// TIA Portal V16 export
// export: Created 2021-11-12T13:31:02.9636744Z, ExportSetting WithDefaults, DisplayName Totally Integrated Automation Portal, DisplayVersion V16 Update 3, DisplayName TIA Portal Version Control Interface, DisplayVersion V16 Update 2, DisplayName TIA Portal Openness, DisplayVersion V16 Update 3, DisplayName SINAMICS Startdrive Advanced, DisplayVersion V16 Update 5, DisplayName SINAMICS Startdrive G130, G150, S120, S150, SINAMICS MV, S210, DisplayVersion V16 Update 5, DisplayName SINAMICS Startdrive G110M, G120, G120C, G120D, G120P, G115D, DisplayVersion V16 Update 5, DisplayName STEP 7 Professional, DisplayVersion V16 Update 3, DisplayName STEP 7 Safety, DisplayVersion V16, DisplayName WinCC UA Professional, DisplayVersion V16 Update 3
FUNCTION_BLOCK "DataColl"   // FB65, LAD
TITLE = Data Collector for SCADA
{ S7_Optimized_Access := 'TRUE' }
VERSION : 0.1
// stored: AutoNumber true, IsIECCheckEnabled false, IsRetainMemResEnabled false, MemoryReserve 100, SetENOAutomatically false, UDAEnableTagReadback false
   VAR
      SS_Edge : Array[0..9] of Bool;
      SF_ArchivePeriodicallyFullAlarm : "STD_DI_Mon";
      SF_ArchivePeriodicallyFullWarn : "STD_DI_Mon";
      SF_ArchiveItemFullAlarm : "STD_DI_Mon";
      SF_ArchiveItemFullWarn : "STD_DI_Mon";
      SF_FIFOQueueArchivePeriodically : "FIFOQueueArchivPeriodically";   // FIFO for data collected periodically
      SF_FIFOQueueArchiveItem : "FIFOQueueArchivItem";   // FIFO for data collected on trigger
      SI_PointerArchivePeriodically : Int;   // Pointer in FIFO
      SI_PointerArchiveItem : Int;   // Pointer in FIFo
      SB1_BufferArchivePeriodicallyFullAlarm : Bool;   // Buffer full alarm
      SB1_BufferArchivePeriodicallyFullWarn : Bool;   // Buffer full warning
      SB1_BufferArchiveItemFullAlarm : Bool;   // Buffer full alarm
      SB1_BufferArchiveItemFullWarn : Bool;   // Buffer full warning
   END_VAR
   VAR_TEMP
      TB1CmdReader_ArchivePeriodically : Bool;   // Command to write data into FIFO
      TB1CmdReader_ArchiveItem1 : Bool;   // Command to write data into FIFO
      TB1CmdReader_ArchiveItem2 : Bool;   // Command to write data into FIFO
      TB1ArchiveItemDone : Bool;   // Writing data to FIFO done
      TB1EnableArchivePeriodically : Bool;   // Enable to archive data periodically
      TI_ArchiveLenght : Int;
   END_VAR
   VAR_TEMP   // added for the SCL form of the ladder/FBD networks
      _w1 : Bool;
      _w2 : Bool;
   END_VAR
BEGIN

REGION Network 1: Clear temporary variables
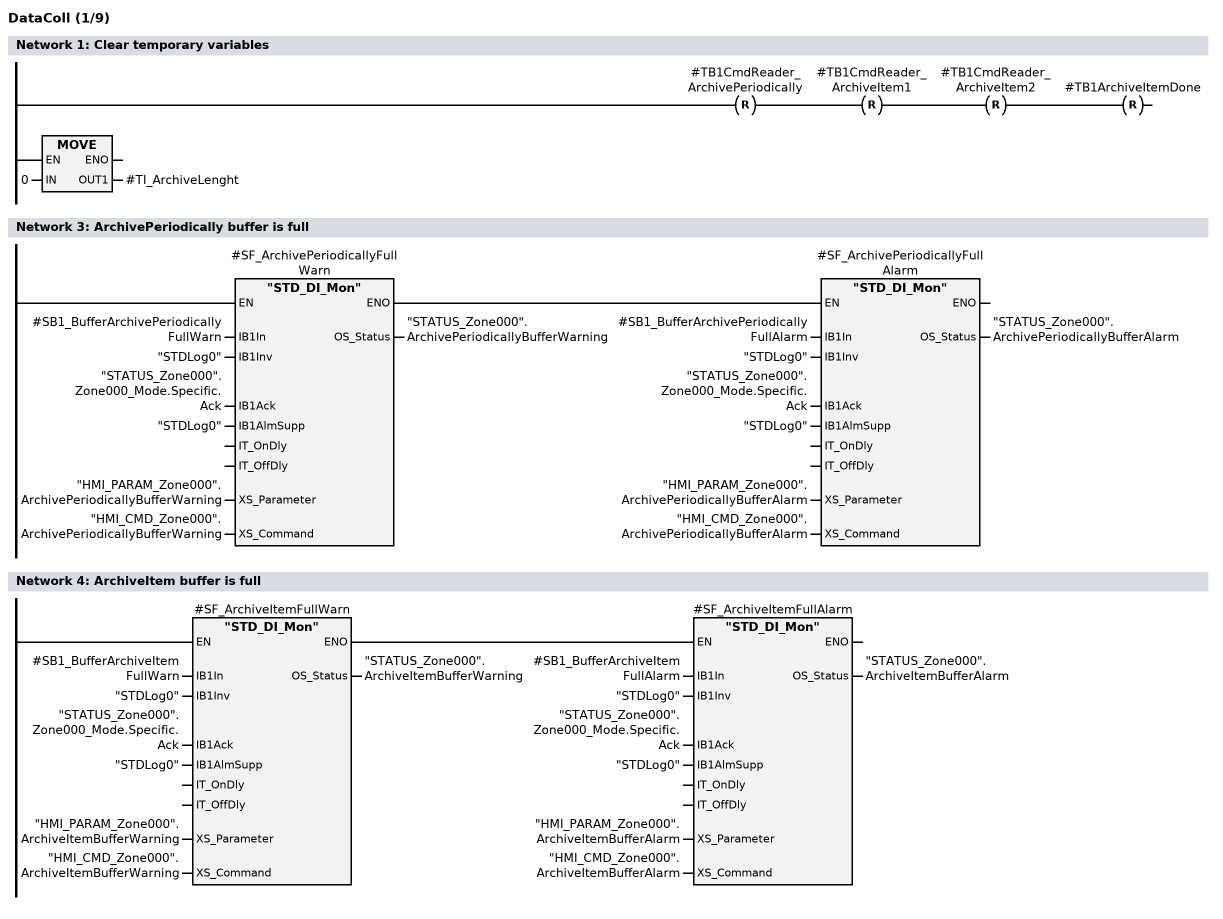
   RUNG wire#powerrail
      R_Coil( #TB1CmdReader_ArchivePeriodically )
      R_Coil( #TB1CmdReader_ArchiveItem1 )
      R_Coil( #TB1CmdReader_ArchiveItem2 )
      R_Coil( #TB1ArchiveItemDone )
   END_RUNG
   RUNG wire#powerrail
      Move(in := 0, out1 => #TI_ArchiveLenght)
   END_RUNG
   // the same network as SCL:
   #TB1CmdReader_ArchivePeriodically := FALSE;
   #TB1CmdReader_ArchiveItem1 := FALSE;
   #TB1CmdReader_ArchiveItem2 := FALSE;
   #TB1ArchiveItemDone := FALSE;
   #TI_ArchiveLenght := 0;
END_REGION

REGION Network 2: *************** Alarms ***************
END_REGION

REGION Network 3: ArchivePeriodically buffer is full
   RUNG wire#powerrail
      #SF_ArchivePeriodicallyFullWarn(IB1In := #SB1_BufferArchivePeriodicallyFullWarn, IB1Inv := "STDLog0", IB1Ack := "STATUS_Zone000".Zone000_Mode.Specific.Ack, IB1AlmSupp := "STDLog0", IT_OnDly :=, IT_OffDly :=, XS_Parameter := "HMI_PARAM_Zone000".ArchivePeriodicallyBufferWarning, XS_Command := "HMI_CMD_Zone000".ArchivePeriodicallyBufferWarning, OS_Status => "STATUS_Zone000".ArchivePeriodicallyBufferWarning)
      #SF_ArchivePeriodicallyFullAlarm(IB1In := #SB1_BufferArchivePeriodicallyFullAlarm, IB1Inv := "STDLog0", IB1Ack := "STATUS_Zone000".Zone000_Mode.Specific.Ack, IB1AlmSupp := "STDLog0", IT_OnDly :=, IT_OffDly :=, XS_Parameter := "HMI_PARAM_Zone000".ArchivePeriodicallyBufferAlarm, XS_Command := "HMI_CMD_Zone000".ArchivePeriodicallyBufferAlarm, OS_Status => "STATUS_Zone000".ArchivePeriodicallyBufferAlarm)
   END_RUNG
   // the same network as SCL:
   #SF_ArchivePeriodicallyFullWarn(IB1In := #SB1_BufferArchivePeriodicallyFullWarn,   // "STD_DI_Mon"
                           IB1Inv := "STDLog0",
                           IB1Ack := "STATUS_Zone000".Zone000_Mode.Specific.Ack,
                           IB1AlmSupp := "STDLog0",
                           XS_Parameter := "HMI_PARAM_Zone000".ArchivePeriodicallyBufferWarning,
                           XS_Command := "HMI_CMD_Zone000".ArchivePeriodicallyBufferWarning,
                           OS_Status => "STATUS_Zone000".ArchivePeriodicallyBufferWarning,
                           ENO => #_w1);
   IF #_w1 THEN
       #SF_ArchivePeriodicallyFullAlarm(IB1In := #SB1_BufferArchivePeriodicallyFullAlarm,   // "STD_DI_Mon"
                               IB1Inv := "STDLog0",
                               IB1Ack := "STATUS_Zone000".Zone000_Mode.Specific.Ack,
                               IB1AlmSupp := "STDLog0",
                               XS_Parameter := "HMI_PARAM_Zone000".ArchivePeriodicallyBufferAlarm,
                               XS_Command := "HMI_CMD_Zone000".ArchivePeriodicallyBufferAlarm,
                               OS_Status => "STATUS_Zone000".ArchivePeriodicallyBufferAlarm);
   END_IF;
END_REGION

REGION Network 4: ArchiveItem buffer is full
   RUNG wire#powerrail
      #SF_ArchiveItemFullWarn(IB1In := #SB1_BufferArchiveItemFullWarn, IB1Inv := "STDLog0", IB1Ack := "STATUS_Zone000".Zone000_Mode.Specific.Ack, IB1AlmSupp := "STDLog0", IT_OnDly :=, IT_OffDly :=, XS_Parameter := "HMI_PARAM_Zone000".ArchiveItemBufferWarning, XS_Command := "HMI_CMD_Zone000".ArchiveItemBufferWarning, OS_Status => "STATUS_Zone000".ArchiveItemBufferWarning)
      #SF_ArchiveItemFullAlarm(IB1In := #SB1_BufferArchiveItemFullAlarm, IB1Inv := "STDLog0", IB1Ack := "STATUS_Zone000".Zone000_Mode.Specific.Ack, IB1AlmSupp := "STDLog0", IT_OnDly :=, IT_OffDly :=, XS_Parameter := "HMI_PARAM_Zone000".ArchiveItemBufferAlarm, XS_Command := "HMI_CMD_Zone000".ArchiveItemBufferAlarm, OS_Status => "STATUS_Zone000".ArchiveItemBufferAlarm)
   END_RUNG
   // the same network as SCL:
   #SF_ArchiveItemFullWarn(IB1In := #SB1_BufferArchiveItemFullWarn,   // "STD_DI_Mon"
                           IB1Inv := "STDLog0",
                           IB1Ack := "STATUS_Zone000".Zone000_Mode.Specific.Ack,
                           IB1AlmSupp := "STDLog0",
                           XS_Parameter := "HMI_PARAM_Zone000".ArchiveItemBufferWarning,
                           XS_Command := "HMI_CMD_Zone000".ArchiveItemBufferWarning,
                           OS_Status => "STATUS_Zone000".ArchiveItemBufferWarning,
                           ENO => #_w1);
   IF #_w1 THEN
       #SF_ArchiveItemFullAlarm(IB1In := #SB1_BufferArchiveItemFullAlarm,   // "STD_DI_Mon"
                               IB1Inv := "STDLog0",
                               IB1Ack := "STATUS_Zone000".Zone000_Mode.Specific.Ack,
                               IB1AlmSupp := "STDLog0",
                               XS_Parameter := "HMI_PARAM_Zone000".ArchiveItemBufferAlarm,
                               XS_Command := "HMI_CMD_Zone000".ArchiveItemBufferAlarm,
                               OS_Status => "STATUS_Zone000".ArchiveItemBufferAlarm);
   END_IF;
END_REGION

REGION Network 5: ************** Data collecting on trigger ***************
END_REGION

REGION Network 6: Filling interface for item1
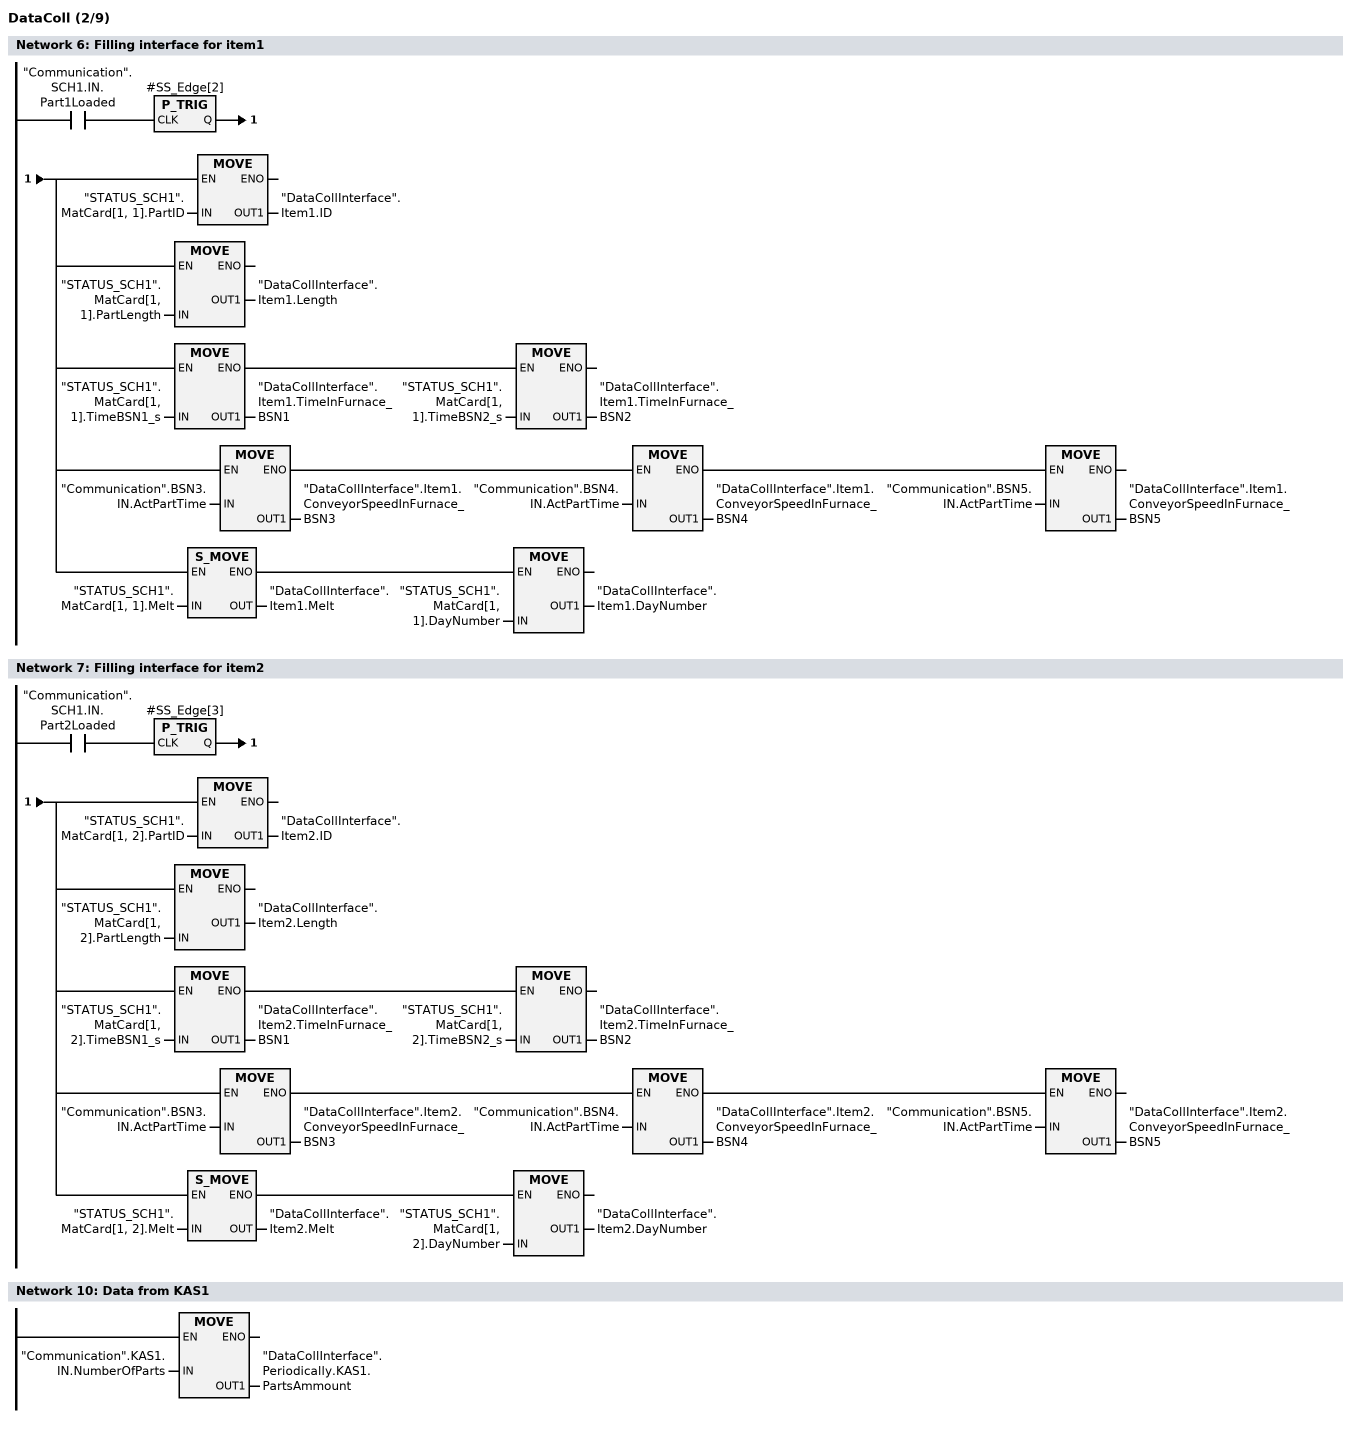
   RUNG wire#powerrail
      Contact( "Communication".SCH1.IN.Part1Loaded )
      P_Trig( #SS_Edge[2] )
      wire#w1
      Move(in := "STATUS_SCH1".MatCard[1, 1].PartID, out1 => "DataCollInterface".Item1.ID)
   END_RUNG
   RUNG wire#w1
      Move(in := "STATUS_SCH1".MatCard[1, 1].PartLength, out1 => "DataCollInterface".Item1.Length)
   END_RUNG
   RUNG wire#w1
      Move(in := "STATUS_SCH1".MatCard[1, 1].TimeBSN1_s, out1 => "DataCollInterface".Item1.TimeInFurnace_BSN1)
      Move(in := "STATUS_SCH1".MatCard[1, 1].TimeBSN2_s, out1 => "DataCollInterface".Item1.TimeInFurnace_BSN2)
   END_RUNG
   RUNG wire#w1
      Move(in := "Communication".BSN3.IN.ActPartTime, out1 => "DataCollInterface".Item1.ConveyorSpeedInFurnace_BSN3)
      Move(in := "Communication".BSN4.IN.ActPartTime, out1 => "DataCollInterface".Item1.ConveyorSpeedInFurnace_BSN4)
      Move(in := "Communication".BSN5.IN.ActPartTime, out1 => "DataCollInterface".Item1.ConveyorSpeedInFurnace_BSN5)
   END_RUNG
   RUNG wire#w1
      S_Move(in := "STATUS_SCH1".MatCard[1, 1].Melt, out => "DataCollInterface".Item1.Melt)
      Move(in := "STATUS_SCH1".MatCard[1, 1].DayNumber, out1 => "DataCollInterface".Item1.DayNumber)
   END_RUNG
   // the same network as SCL:
   #_w1 := "Communication".SCH1.IN.Part1Loaded AND NOT #SS_Edge[2];   // rising edge
   #SS_Edge[2] := "Communication".SCH1.IN.Part1Loaded;
   IF #_w1 THEN
       "DataCollInterface".Item1.ID := "STATUS_SCH1".MatCard[1, 1].PartID;
       "DataCollInterface".Item1.Length := "STATUS_SCH1".MatCard[1, 1].PartLength;
       "DataCollInterface".Item1.TimeInFurnace_BSN1 := "STATUS_SCH1".MatCard[1, 1].TimeBSN1_s;
       "DataCollInterface".Item1.TimeInFurnace_BSN2 := "STATUS_SCH1".MatCard[1, 1].TimeBSN2_s;
       "DataCollInterface".Item1.ConveyorSpeedInFurnace_BSN3 := "Communication".BSN3.IN.ActPartTime;
       "DataCollInterface".Item1.ConveyorSpeedInFurnace_BSN4 := "Communication".BSN4.IN.ActPartTime;
       "DataCollInterface".Item1.ConveyorSpeedInFurnace_BSN5 := "Communication".BSN5.IN.ActPartTime;
       "DataCollInterface".Item1.Melt := "STATUS_SCH1".MatCard[1, 1].Melt;
       "DataCollInterface".Item1.DayNumber := "STATUS_SCH1".MatCard[1, 1].DayNumber;
   END_IF;
END_REGION

REGION Network 7: Filling interface for item2
   RUNG wire#powerrail
      Contact( "Communication".SCH1.IN.Part2Loaded )
      P_Trig( #SS_Edge[3] )
      wire#w1
      Move(in := "STATUS_SCH1".MatCard[1, 2].PartID, out1 => "DataCollInterface".Item2.ID)
   END_RUNG
   RUNG wire#w1
      Move(in := "STATUS_SCH1".MatCard[1, 2].PartLength, out1 => "DataCollInterface".Item2.Length)
   END_RUNG
   RUNG wire#w1
      Move(in := "STATUS_SCH1".MatCard[1, 2].TimeBSN1_s, out1 => "DataCollInterface".Item2.TimeInFurnace_BSN1)
      Move(in := "STATUS_SCH1".MatCard[1, 2].TimeBSN2_s, out1 => "DataCollInterface".Item2.TimeInFurnace_BSN2)
   END_RUNG
   RUNG wire#w1
      Move(in := "Communication".BSN3.IN.ActPartTime, out1 => "DataCollInterface".Item2.ConveyorSpeedInFurnace_BSN3)
      Move(in := "Communication".BSN4.IN.ActPartTime, out1 => "DataCollInterface".Item2.ConveyorSpeedInFurnace_BSN4)
      Move(in := "Communication".BSN5.IN.ActPartTime, out1 => "DataCollInterface".Item2.ConveyorSpeedInFurnace_BSN5)
   END_RUNG
   RUNG wire#w1
      S_Move(in := "STATUS_SCH1".MatCard[1, 2].Melt, out => "DataCollInterface".Item2.Melt)
      Move(in := "STATUS_SCH1".MatCard[1, 2].DayNumber, out1 => "DataCollInterface".Item2.DayNumber)
   END_RUNG
   // the same network as SCL:
   #_w1 := "Communication".SCH1.IN.Part2Loaded AND NOT #SS_Edge[3];   // rising edge
   #SS_Edge[3] := "Communication".SCH1.IN.Part2Loaded;
   IF #_w1 THEN
       "DataCollInterface".Item2.ID := "STATUS_SCH1".MatCard[1, 2].PartID;
       "DataCollInterface".Item2.Length := "STATUS_SCH1".MatCard[1, 2].PartLength;
       "DataCollInterface".Item2.TimeInFurnace_BSN1 := "STATUS_SCH1".MatCard[1, 2].TimeBSN1_s;
       "DataCollInterface".Item2.TimeInFurnace_BSN2 := "STATUS_SCH1".MatCard[1, 2].TimeBSN2_s;
       "DataCollInterface".Item2.ConveyorSpeedInFurnace_BSN3 := "Communication".BSN3.IN.ActPartTime;
       "DataCollInterface".Item2.ConveyorSpeedInFurnace_BSN4 := "Communication".BSN4.IN.ActPartTime;
       "DataCollInterface".Item2.ConveyorSpeedInFurnace_BSN5 := "Communication".BSN5.IN.ActPartTime;
       "DataCollInterface".Item2.Melt := "STATUS_SCH1".MatCard[1, 2].Melt;
       "DataCollInterface".Item2.DayNumber := "STATUS_SCH1".MatCard[1, 2].DayNumber;
   END_IF;
END_REGION

REGION Network 8: ************** Data collecting periodically ***************
END_REGION

REGION Network 9: ************** Saws ***************
END_REGION

REGION Network 10: Data from KAS1
   RUNG wire#powerrail
      Move(in := "Communication".KAS1.IN.NumberOfParts, out1 => "DataCollInterface".Periodically.KAS1.PartsAmmount)
   END_RUNG
   // the same network as SCL:
   "DataCollInterface".Periodically.KAS1.PartsAmmount := "Communication".KAS1.IN.NumberOfParts;
END_REGION

REGION Network 11: Data from KAS2
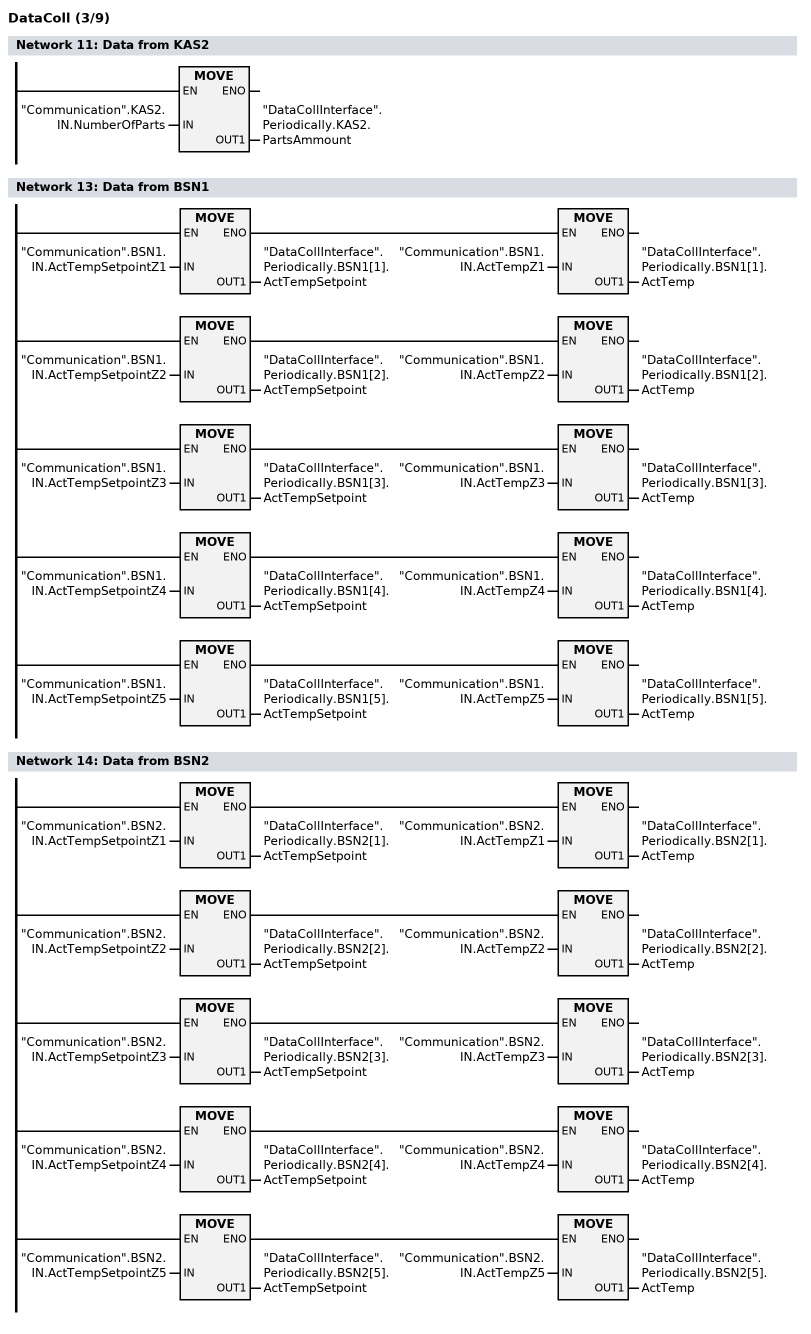
   RUNG wire#powerrail
      Move(in := "Communication".KAS2.IN.NumberOfParts, out1 => "DataCollInterface".Periodically.KAS2.PartsAmmount)
   END_RUNG
   // the same network as SCL:
   "DataCollInterface".Periodically.KAS2.PartsAmmount := "Communication".KAS2.IN.NumberOfParts;
END_REGION

REGION Network 12: ***************Owens ***************
END_REGION

REGION Network 13: Data from BSN1
   RUNG wire#powerrail
      Move(in := "Communication".BSN1.IN.ActTempSetpointZ1, out1 => "DataCollInterface".Periodically.BSN1[1].ActTempSetpoint)
      Move(in := "Communication".BSN1.IN.ActTempZ1, out1 => "DataCollInterface".Periodically.BSN1[1].ActTemp)
   END_RUNG
   RUNG wire#powerrail
      Move(in := "Communication".BSN1.IN.ActTempSetpointZ2, out1 => "DataCollInterface".Periodically.BSN1[2].ActTempSetpoint)
      Move(in := "Communication".BSN1.IN.ActTempZ2, out1 => "DataCollInterface".Periodically.BSN1[2].ActTemp)
   END_RUNG
   RUNG wire#powerrail
      Move(in := "Communication".BSN1.IN.ActTempSetpointZ3, out1 => "DataCollInterface".Periodically.BSN1[3].ActTempSetpoint)
      Move(in := "Communication".BSN1.IN.ActTempZ3, out1 => "DataCollInterface".Periodically.BSN1[3].ActTemp)
   END_RUNG
   RUNG wire#powerrail
      Move(in := "Communication".BSN1.IN.ActTempSetpointZ4, out1 => "DataCollInterface".Periodically.BSN1[4].ActTempSetpoint)
      Move(in := "Communication".BSN1.IN.ActTempZ4, out1 => "DataCollInterface".Periodically.BSN1[4].ActTemp)
   END_RUNG
   RUNG wire#powerrail
      Move(in := "Communication".BSN1.IN.ActTempSetpointZ5, out1 => "DataCollInterface".Periodically.BSN1[5].ActTempSetpoint)
      Move(in := "Communication".BSN1.IN.ActTempZ5, out1 => "DataCollInterface".Periodically.BSN1[5].ActTemp)
   END_RUNG
   // the same network as SCL:
   "DataCollInterface".Periodically.BSN1[1].ActTempSetpoint := "Communication".BSN1.IN.ActTempSetpointZ1;
   "DataCollInterface".Periodically.BSN1[1].ActTemp := "Communication".BSN1.IN.ActTempZ1;
   "DataCollInterface".Periodically.BSN1[2].ActTempSetpoint := "Communication".BSN1.IN.ActTempSetpointZ2;
   "DataCollInterface".Periodically.BSN1[2].ActTemp := "Communication".BSN1.IN.ActTempZ2;
   "DataCollInterface".Periodically.BSN1[3].ActTempSetpoint := "Communication".BSN1.IN.ActTempSetpointZ3;
   "DataCollInterface".Periodically.BSN1[3].ActTemp := "Communication".BSN1.IN.ActTempZ3;
   "DataCollInterface".Periodically.BSN1[4].ActTempSetpoint := "Communication".BSN1.IN.ActTempSetpointZ4;
   "DataCollInterface".Periodically.BSN1[4].ActTemp := "Communication".BSN1.IN.ActTempZ4;
   "DataCollInterface".Periodically.BSN1[5].ActTempSetpoint := "Communication".BSN1.IN.ActTempSetpointZ5;
   "DataCollInterface".Periodically.BSN1[5].ActTemp := "Communication".BSN1.IN.ActTempZ5;
END_REGION

REGION Network 14: Data from BSN2
   RUNG wire#powerrail
      Move(in := "Communication".BSN2.IN.ActTempSetpointZ1, out1 => "DataCollInterface".Periodically.BSN2[1].ActTempSetpoint)
      Move(in := "Communication".BSN2.IN.ActTempZ1, out1 => "DataCollInterface".Periodically.BSN2[1].ActTemp)
   END_RUNG
   RUNG wire#powerrail
      Move(in := "Communication".BSN2.IN.ActTempSetpointZ2, out1 => "DataCollInterface".Periodically.BSN2[2].ActTempSetpoint)
      Move(in := "Communication".BSN2.IN.ActTempZ2, out1 => "DataCollInterface".Periodically.BSN2[2].ActTemp)
   END_RUNG
   RUNG wire#powerrail
      Move(in := "Communication".BSN2.IN.ActTempSetpointZ3, out1 => "DataCollInterface".Periodically.BSN2[3].ActTempSetpoint)
      Move(in := "Communication".BSN2.IN.ActTempZ3, out1 => "DataCollInterface".Periodically.BSN2[3].ActTemp)
   END_RUNG
   RUNG wire#powerrail
      Move(in := "Communication".BSN2.IN.ActTempSetpointZ4, out1 => "DataCollInterface".Periodically.BSN2[4].ActTempSetpoint)
      Move(in := "Communication".BSN2.IN.ActTempZ4, out1 => "DataCollInterface".Periodically.BSN2[4].ActTemp)
   END_RUNG
   RUNG wire#powerrail
      Move(in := "Communication".BSN2.IN.ActTempSetpointZ5, out1 => "DataCollInterface".Periodically.BSN2[5].ActTempSetpoint)
      Move(in := "Communication".BSN2.IN.ActTempZ5, out1 => "DataCollInterface".Periodically.BSN2[5].ActTemp)
   END_RUNG
   // the same network as SCL:
   "DataCollInterface".Periodically.BSN2[1].ActTempSetpoint := "Communication".BSN2.IN.ActTempSetpointZ1;
   "DataCollInterface".Periodically.BSN2[1].ActTemp := "Communication".BSN2.IN.ActTempZ1;
   "DataCollInterface".Periodically.BSN2[2].ActTempSetpoint := "Communication".BSN2.IN.ActTempSetpointZ2;
   "DataCollInterface".Periodically.BSN2[2].ActTemp := "Communication".BSN2.IN.ActTempZ2;
   "DataCollInterface".Periodically.BSN2[3].ActTempSetpoint := "Communication".BSN2.IN.ActTempSetpointZ3;
   "DataCollInterface".Periodically.BSN2[3].ActTemp := "Communication".BSN2.IN.ActTempZ3;
   "DataCollInterface".Periodically.BSN2[4].ActTempSetpoint := "Communication".BSN2.IN.ActTempSetpointZ4;
   "DataCollInterface".Periodically.BSN2[4].ActTemp := "Communication".BSN2.IN.ActTempZ4;
   "DataCollInterface".Periodically.BSN2[5].ActTempSetpoint := "Communication".BSN2.IN.ActTempSetpointZ5;
   "DataCollInterface".Periodically.BSN2[5].ActTemp := "Communication".BSN2.IN.ActTempZ5;
END_REGION

REGION Network 15: Data from BSN3
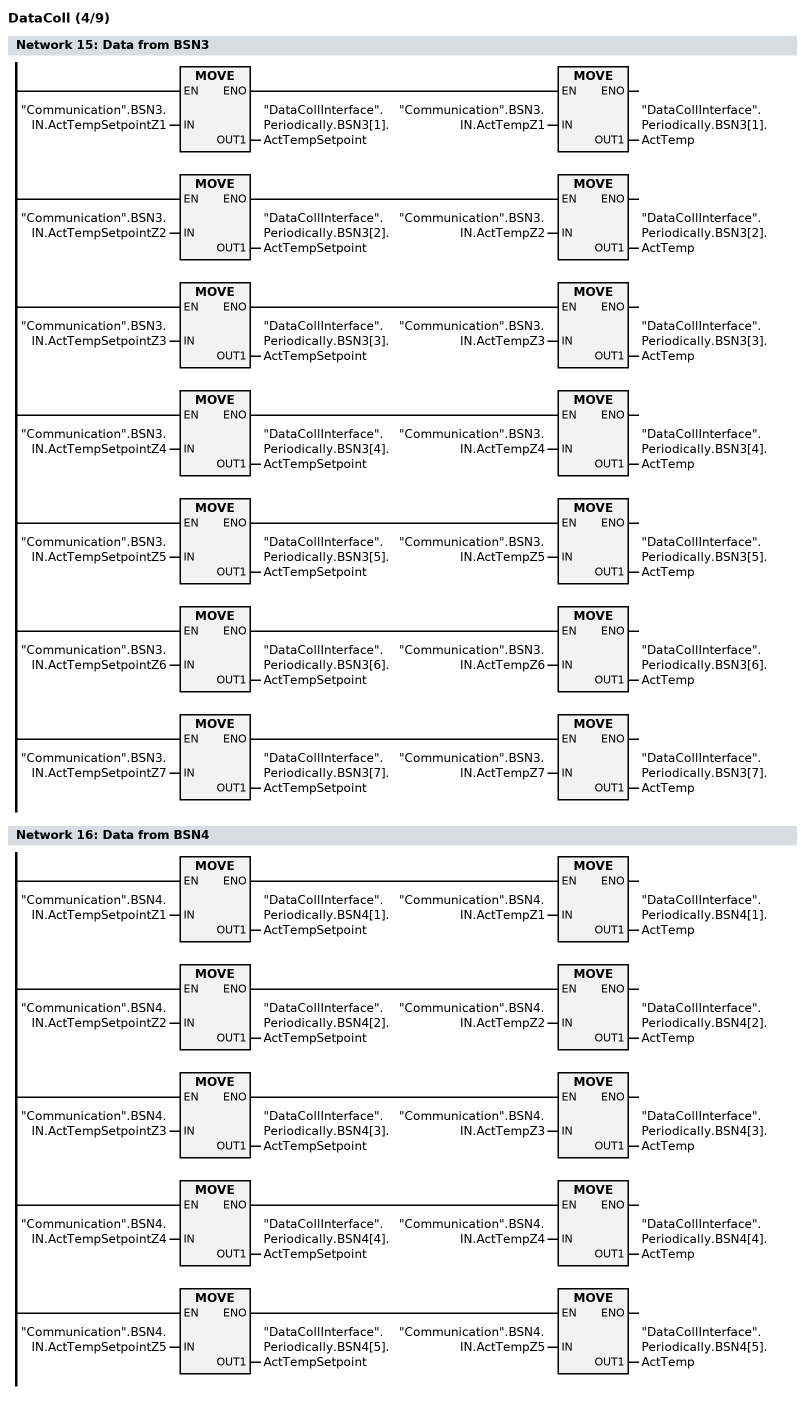
   RUNG wire#powerrail
      Move(in := "Communication".BSN3.IN.ActTempSetpointZ1, out1 => "DataCollInterface".Periodically.BSN3[1].ActTempSetpoint)
      Move(in := "Communication".BSN3.IN.ActTempZ1, out1 => "DataCollInterface".Periodically.BSN3[1].ActTemp)
   END_RUNG
   RUNG wire#powerrail
      Move(in := "Communication".BSN3.IN.ActTempSetpointZ2, out1 => "DataCollInterface".Periodically.BSN3[2].ActTempSetpoint)
      Move(in := "Communication".BSN3.IN.ActTempZ2, out1 => "DataCollInterface".Periodically.BSN3[2].ActTemp)
   END_RUNG
   RUNG wire#powerrail
      Move(in := "Communication".BSN3.IN.ActTempSetpointZ3, out1 => "DataCollInterface".Periodically.BSN3[3].ActTempSetpoint)
      Move(in := "Communication".BSN3.IN.ActTempZ3, out1 => "DataCollInterface".Periodically.BSN3[3].ActTemp)
   END_RUNG
   RUNG wire#powerrail
      Move(in := "Communication".BSN3.IN.ActTempSetpointZ4, out1 => "DataCollInterface".Periodically.BSN3[4].ActTempSetpoint)
      Move(in := "Communication".BSN3.IN.ActTempZ4, out1 => "DataCollInterface".Periodically.BSN3[4].ActTemp)
   END_RUNG
   RUNG wire#powerrail
      Move(in := "Communication".BSN3.IN.ActTempSetpointZ5, out1 => "DataCollInterface".Periodically.BSN3[5].ActTempSetpoint)
      Move(in := "Communication".BSN3.IN.ActTempZ5, out1 => "DataCollInterface".Periodically.BSN3[5].ActTemp)
   END_RUNG
   RUNG wire#powerrail
      Move(in := "Communication".BSN3.IN.ActTempSetpointZ6, out1 => "DataCollInterface".Periodically.BSN3[6].ActTempSetpoint)
      Move(in := "Communication".BSN3.IN.ActTempZ6, out1 => "DataCollInterface".Periodically.BSN3[6].ActTemp)
   END_RUNG
   RUNG wire#powerrail
      Move(in := "Communication".BSN3.IN.ActTempSetpointZ7, out1 => "DataCollInterface".Periodically.BSN3[7].ActTempSetpoint)
      Move(in := "Communication".BSN3.IN.ActTempZ7, out1 => "DataCollInterface".Periodically.BSN3[7].ActTemp)
   END_RUNG
   // the same network as SCL:
   "DataCollInterface".Periodically.BSN3[1].ActTempSetpoint := "Communication".BSN3.IN.ActTempSetpointZ1;
   "DataCollInterface".Periodically.BSN3[1].ActTemp := "Communication".BSN3.IN.ActTempZ1;
   "DataCollInterface".Periodically.BSN3[2].ActTempSetpoint := "Communication".BSN3.IN.ActTempSetpointZ2;
   "DataCollInterface".Periodically.BSN3[2].ActTemp := "Communication".BSN3.IN.ActTempZ2;
   "DataCollInterface".Periodically.BSN3[3].ActTempSetpoint := "Communication".BSN3.IN.ActTempSetpointZ3;
   "DataCollInterface".Periodically.BSN3[3].ActTemp := "Communication".BSN3.IN.ActTempZ3;
   "DataCollInterface".Periodically.BSN3[4].ActTempSetpoint := "Communication".BSN3.IN.ActTempSetpointZ4;
   "DataCollInterface".Periodically.BSN3[4].ActTemp := "Communication".BSN3.IN.ActTempZ4;
   "DataCollInterface".Periodically.BSN3[5].ActTempSetpoint := "Communication".BSN3.IN.ActTempSetpointZ5;
   "DataCollInterface".Periodically.BSN3[5].ActTemp := "Communication".BSN3.IN.ActTempZ5;
   "DataCollInterface".Periodically.BSN3[6].ActTempSetpoint := "Communication".BSN3.IN.ActTempSetpointZ6;
   "DataCollInterface".Periodically.BSN3[6].ActTemp := "Communication".BSN3.IN.ActTempZ6;
   "DataCollInterface".Periodically.BSN3[7].ActTempSetpoint := "Communication".BSN3.IN.ActTempSetpointZ7;
   "DataCollInterface".Periodically.BSN3[7].ActTemp := "Communication".BSN3.IN.ActTempZ7;
END_REGION

REGION Network 16: Data from BSN4
   RUNG wire#powerrail
      Move(in := "Communication".BSN4.IN.ActTempSetpointZ1, out1 => "DataCollInterface".Periodically.BSN4[1].ActTempSetpoint)
      Move(in := "Communication".BSN4.IN.ActTempZ1, out1 => "DataCollInterface".Periodically.BSN4[1].ActTemp)
   END_RUNG
   RUNG wire#powerrail
      Move(in := "Communication".BSN4.IN.ActTempSetpointZ2, out1 => "DataCollInterface".Periodically.BSN4[2].ActTempSetpoint)
      Move(in := "Communication".BSN4.IN.ActTempZ2, out1 => "DataCollInterface".Periodically.BSN4[2].ActTemp)
   END_RUNG
   RUNG wire#powerrail
      Move(in := "Communication".BSN4.IN.ActTempSetpointZ3, out1 => "DataCollInterface".Periodically.BSN4[3].ActTempSetpoint)
      Move(in := "Communication".BSN4.IN.ActTempZ3, out1 => "DataCollInterface".Periodically.BSN4[3].ActTemp)
   END_RUNG
   RUNG wire#powerrail
      Move(in := "Communication".BSN4.IN.ActTempSetpointZ4, out1 => "DataCollInterface".Periodically.BSN4[4].ActTempSetpoint)
      Move(in := "Communication".BSN4.IN.ActTempZ4, out1 => "DataCollInterface".Periodically.BSN4[4].ActTemp)
   END_RUNG
   RUNG wire#powerrail
      Move(in := "Communication".BSN4.IN.ActTempSetpointZ5, out1 => "DataCollInterface".Periodically.BSN4[5].ActTempSetpoint)
      Move(in := "Communication".BSN4.IN.ActTempZ5, out1 => "DataCollInterface".Periodically.BSN4[5].ActTemp)
   END_RUNG
   // the same network as SCL:
   "DataCollInterface".Periodically.BSN4[1].ActTempSetpoint := "Communication".BSN4.IN.ActTempSetpointZ1;
   "DataCollInterface".Periodically.BSN4[1].ActTemp := "Communication".BSN4.IN.ActTempZ1;
   "DataCollInterface".Periodically.BSN4[2].ActTempSetpoint := "Communication".BSN4.IN.ActTempSetpointZ2;
   "DataCollInterface".Periodically.BSN4[2].ActTemp := "Communication".BSN4.IN.ActTempZ2;
   "DataCollInterface".Periodically.BSN4[3].ActTempSetpoint := "Communication".BSN4.IN.ActTempSetpointZ3;
   "DataCollInterface".Periodically.BSN4[3].ActTemp := "Communication".BSN4.IN.ActTempZ3;
   "DataCollInterface".Periodically.BSN4[4].ActTempSetpoint := "Communication".BSN4.IN.ActTempSetpointZ4;
   "DataCollInterface".Periodically.BSN4[4].ActTemp := "Communication".BSN4.IN.ActTempZ4;
   "DataCollInterface".Periodically.BSN4[5].ActTempSetpoint := "Communication".BSN4.IN.ActTempSetpointZ5;
   "DataCollInterface".Periodically.BSN4[5].ActTemp := "Communication".BSN4.IN.ActTempZ5;
END_REGION

REGION Network 17: Data from BSN5
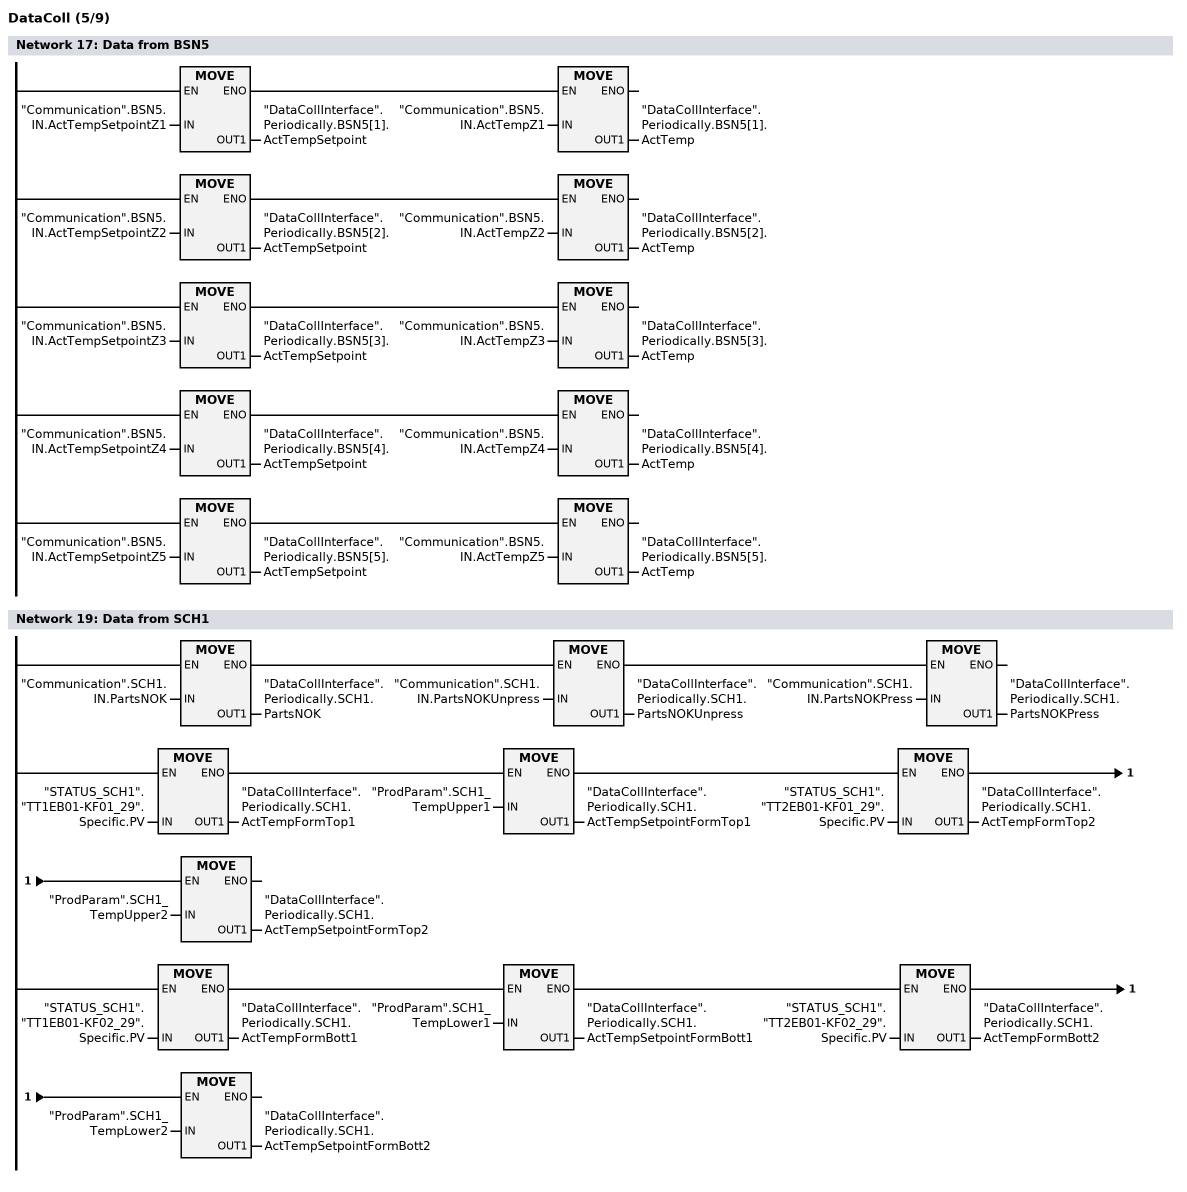
   RUNG wire#powerrail
      Move(in := "Communication".BSN5.IN.ActTempSetpointZ1, out1 => "DataCollInterface".Periodically.BSN5[1].ActTempSetpoint)
      Move(in := "Communication".BSN5.IN.ActTempZ1, out1 => "DataCollInterface".Periodically.BSN5[1].ActTemp)
   END_RUNG
   RUNG wire#powerrail
      Move(in := "Communication".BSN5.IN.ActTempSetpointZ2, out1 => "DataCollInterface".Periodically.BSN5[2].ActTempSetpoint)
      Move(in := "Communication".BSN5.IN.ActTempZ2, out1 => "DataCollInterface".Periodically.BSN5[2].ActTemp)
   END_RUNG
   RUNG wire#powerrail
      Move(in := "Communication".BSN5.IN.ActTempSetpointZ3, out1 => "DataCollInterface".Periodically.BSN5[3].ActTempSetpoint)
      Move(in := "Communication".BSN5.IN.ActTempZ3, out1 => "DataCollInterface".Periodically.BSN5[3].ActTemp)
   END_RUNG
   RUNG wire#powerrail
      Move(in := "Communication".BSN5.IN.ActTempSetpointZ4, out1 => "DataCollInterface".Periodically.BSN5[4].ActTempSetpoint)
      Move(in := "Communication".BSN5.IN.ActTempZ4, out1 => "DataCollInterface".Periodically.BSN5[4].ActTemp)
   END_RUNG
   RUNG wire#powerrail
      Move(in := "Communication".BSN5.IN.ActTempSetpointZ5, out1 => "DataCollInterface".Periodically.BSN5[5].ActTempSetpoint)
      Move(in := "Communication".BSN5.IN.ActTempZ5, out1 => "DataCollInterface".Periodically.BSN5[5].ActTemp)
   END_RUNG
   // the same network as SCL:
   "DataCollInterface".Periodically.BSN5[1].ActTempSetpoint := "Communication".BSN5.IN.ActTempSetpointZ1;
   "DataCollInterface".Periodically.BSN5[1].ActTemp := "Communication".BSN5.IN.ActTempZ1;
   "DataCollInterface".Periodically.BSN5[2].ActTempSetpoint := "Communication".BSN5.IN.ActTempSetpointZ2;
   "DataCollInterface".Periodically.BSN5[2].ActTemp := "Communication".BSN5.IN.ActTempZ2;
   "DataCollInterface".Periodically.BSN5[3].ActTempSetpoint := "Communication".BSN5.IN.ActTempSetpointZ3;
   "DataCollInterface".Periodically.BSN5[3].ActTemp := "Communication".BSN5.IN.ActTempZ3;
   "DataCollInterface".Periodically.BSN5[4].ActTempSetpoint := "Communication".BSN5.IN.ActTempSetpointZ4;
   "DataCollInterface".Periodically.BSN5[4].ActTemp := "Communication".BSN5.IN.ActTempZ4;
   "DataCollInterface".Periodically.BSN5[5].ActTempSetpoint := "Communication".BSN5.IN.ActTempSetpointZ5;
   "DataCollInterface".Periodically.BSN5[5].ActTemp := "Communication".BSN5.IN.ActTempZ5;
END_REGION

REGION Network 18: *************** Press ***************
END_REGION

REGION Network 19: Data from SCH1
   RUNG wire#powerrail
      Move(in := "Communication".SCH1.IN.PartsNOK, out1 => "DataCollInterface".Periodically.SCH1.PartsNOK)
      Move(in := "Communication".SCH1.IN.PartsNOKUnpress, out1 => "DataCollInterface".Periodically.SCH1.PartsNOKUnpress)
      Move(in := "Communication".SCH1.IN.PartsNOKPress, out1 => "DataCollInterface".Periodically.SCH1.PartsNOKPress)
   END_RUNG
   RUNG wire#powerrail
      Move(in := "STATUS_SCH1"."TT1EB01-KF01_29".Specific.PV, out1 => "DataCollInterface".Periodically.SCH1.ActTempFormTop1)
      Move(in := "ProdParam".SCH1_TempUpper1, out1 => "DataCollInterface".Periodically.SCH1.ActTempSetpointFormTop1)
      Move(in := "STATUS_SCH1"."TT2EB01-KF01_29".Specific.PV, out1 => "DataCollInterface".Periodically.SCH1.ActTempFormTop2)
      Move(in := "ProdParam".SCH1_TempUpper2, out1 => "DataCollInterface".Periodically.SCH1.ActTempSetpointFormTop2)
   END_RUNG
   RUNG wire#powerrail
      Move(in := "STATUS_SCH1"."TT1EB01-KF02_29".Specific.PV, out1 => "DataCollInterface".Periodically.SCH1.ActTempFormBott1)
      Move(in := "ProdParam".SCH1_TempLower1, out1 => "DataCollInterface".Periodically.SCH1.ActTempSetpointFormBott1)
      Move(in := "STATUS_SCH1"."TT2EB01-KF02_29".Specific.PV, out1 => "DataCollInterface".Periodically.SCH1.ActTempFormBott2)
      Move(in := "ProdParam".SCH1_TempLower2, out1 => "DataCollInterface".Periodically.SCH1.ActTempSetpointFormBott2)
   END_RUNG
   // the same network as SCL:
   "DataCollInterface".Periodically.SCH1.PartsNOK := "Communication".SCH1.IN.PartsNOK;
   "DataCollInterface".Periodically.SCH1.PartsNOKUnpress := "Communication".SCH1.IN.PartsNOKUnpress;
   "DataCollInterface".Periodically.SCH1.PartsNOKPress := "Communication".SCH1.IN.PartsNOKPress;
   "DataCollInterface".Periodically.SCH1.ActTempFormTop1 := "STATUS_SCH1"."TT1EB01-KF01_29".Specific.PV;
   "DataCollInterface".Periodically.SCH1.ActTempSetpointFormTop1 := "ProdParam".SCH1_TempUpper1;
   "DataCollInterface".Periodically.SCH1.ActTempFormTop2 := "STATUS_SCH1"."TT2EB01-KF01_29".Specific.PV;
   "DataCollInterface".Periodically.SCH1.ActTempSetpointFormTop2 := "ProdParam".SCH1_TempUpper2;
   "DataCollInterface".Periodically.SCH1.ActTempFormBott1 := "STATUS_SCH1"."TT1EB01-KF02_29".Specific.PV;
   "DataCollInterface".Periodically.SCH1.ActTempSetpointFormBott1 := "ProdParam".SCH1_TempLower1;
   "DataCollInterface".Periodically.SCH1.ActTempFormBott2 := "STATUS_SCH1"."TT2EB01-KF02_29".Specific.PV;
   "DataCollInterface".Periodically.SCH1.ActTempSetpointFormBott2 := "ProdParam".SCH1_TempLower2;
END_REGION

REGION Network 20: *************** Bath ***************
END_REGION

REGION Network 21: Data from 310EQ01
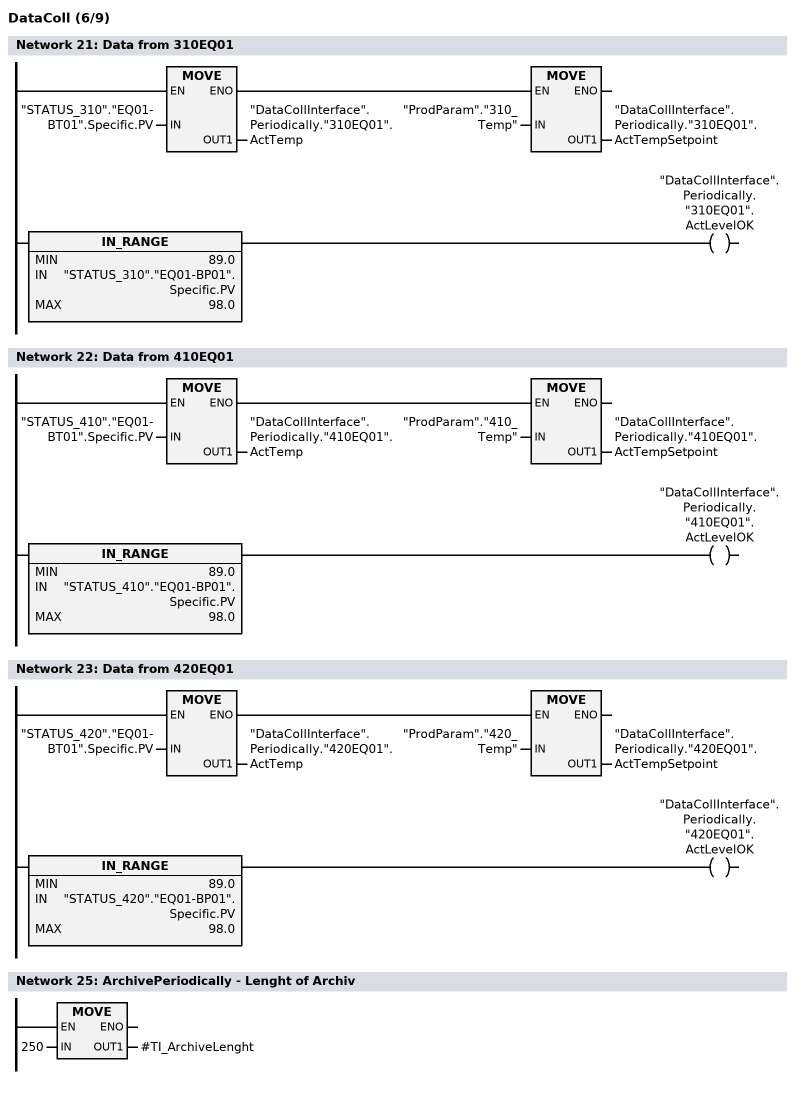
   RUNG wire#powerrail
      Move(in := "STATUS_310"."EQ01-BT01".Specific.PV, out1 => "DataCollInterface".Periodically."310EQ01".ActTemp)
      Move(in := "ProdParam"."310_Temp", out1 => "DataCollInterface".Periodically."310EQ01".ActTempSetpoint)
   END_RUNG
   RUNG wire#powerrail
      { S7_Templates := "SrcType := Real" } InRange(min := 89.0, in := "STATUS_310"."EQ01-BP01".Specific.PV, max := 98.0)
      Coil( "DataCollInterface".Periodically."310EQ01".ActLevelOK )
   END_RUNG
   // the same network as SCL:
   "DataCollInterface".Periodically."310EQ01".ActTemp := "STATUS_310"."EQ01-BT01".Specific.PV;
   "DataCollInterface".Periodically."310EQ01".ActTempSetpoint := "ProdParam"."310_Temp";
   "DataCollInterface".Periodically."310EQ01".ActLevelOK := (89.0 <= "STATUS_310"."EQ01-BP01".Specific.PV) AND ("STATUS_310"."EQ01-BP01".Specific.PV <= 98.0);
END_REGION

REGION Network 22: Data from 410EQ01
   RUNG wire#powerrail
      Move(in := "STATUS_410"."EQ01-BT01".Specific.PV, out1 => "DataCollInterface".Periodically."410EQ01".ActTemp)
      Move(in := "ProdParam"."410_Temp", out1 => "DataCollInterface".Periodically."410EQ01".ActTempSetpoint)
   END_RUNG
   RUNG wire#powerrail
      { S7_Templates := "SrcType := Real" } InRange(min := 89.0, in := "STATUS_410"."EQ01-BP01".Specific.PV, max := 98.0)
      Coil( "DataCollInterface".Periodically."410EQ01".ActLevelOK )
   END_RUNG
   // the same network as SCL:
   "DataCollInterface".Periodically."410EQ01".ActTemp := "STATUS_410"."EQ01-BT01".Specific.PV;
   "DataCollInterface".Periodically."410EQ01".ActTempSetpoint := "ProdParam"."410_Temp";
   "DataCollInterface".Periodically."410EQ01".ActLevelOK := (89.0 <= "STATUS_410"."EQ01-BP01".Specific.PV) AND ("STATUS_410"."EQ01-BP01".Specific.PV <= 98.0);
END_REGION

REGION Network 23: Data from 420EQ01
   RUNG wire#powerrail
      Move(in := "STATUS_420"."EQ01-BT01".Specific.PV, out1 => "DataCollInterface".Periodically."420EQ01".ActTemp)
      Move(in := "ProdParam"."420_Temp", out1 => "DataCollInterface".Periodically."420EQ01".ActTempSetpoint)
   END_RUNG
   RUNG wire#powerrail
      { S7_Templates := "SrcType := Real" } InRange(min := 89.0, in := "STATUS_420"."EQ01-BP01".Specific.PV, max := 98.0)
      Coil( "DataCollInterface".Periodically."420EQ01".ActLevelOK )
   END_RUNG
   // the same network as SCL:
   "DataCollInterface".Periodically."420EQ01".ActTemp := "STATUS_420"."EQ01-BT01".Specific.PV;
   "DataCollInterface".Periodically."420EQ01".ActTempSetpoint := "ProdParam"."420_Temp";
   "DataCollInterface".Periodically."420EQ01".ActLevelOK := (89.0 <= "STATUS_420"."EQ01-BP01".Specific.PV) AND ("STATUS_420"."EQ01-BP01".Specific.PV <= 98.0);
END_REGION

REGION Network 24: *************** ArchivePeriodically ***************
END_REGION

REGION Network 25: ArchivePeriodically - Lenght of Archiv
   RUNG wire#powerrail
      Move(in := 250, out1 => #TI_ArchiveLenght)
   END_RUNG
   // the same network as SCL:
   #TI_ArchiveLenght := 250;
END_REGION

REGION Network 26: Enable to archive data periodically
   // "JSA0Comm" - pritomnost kusu v linke
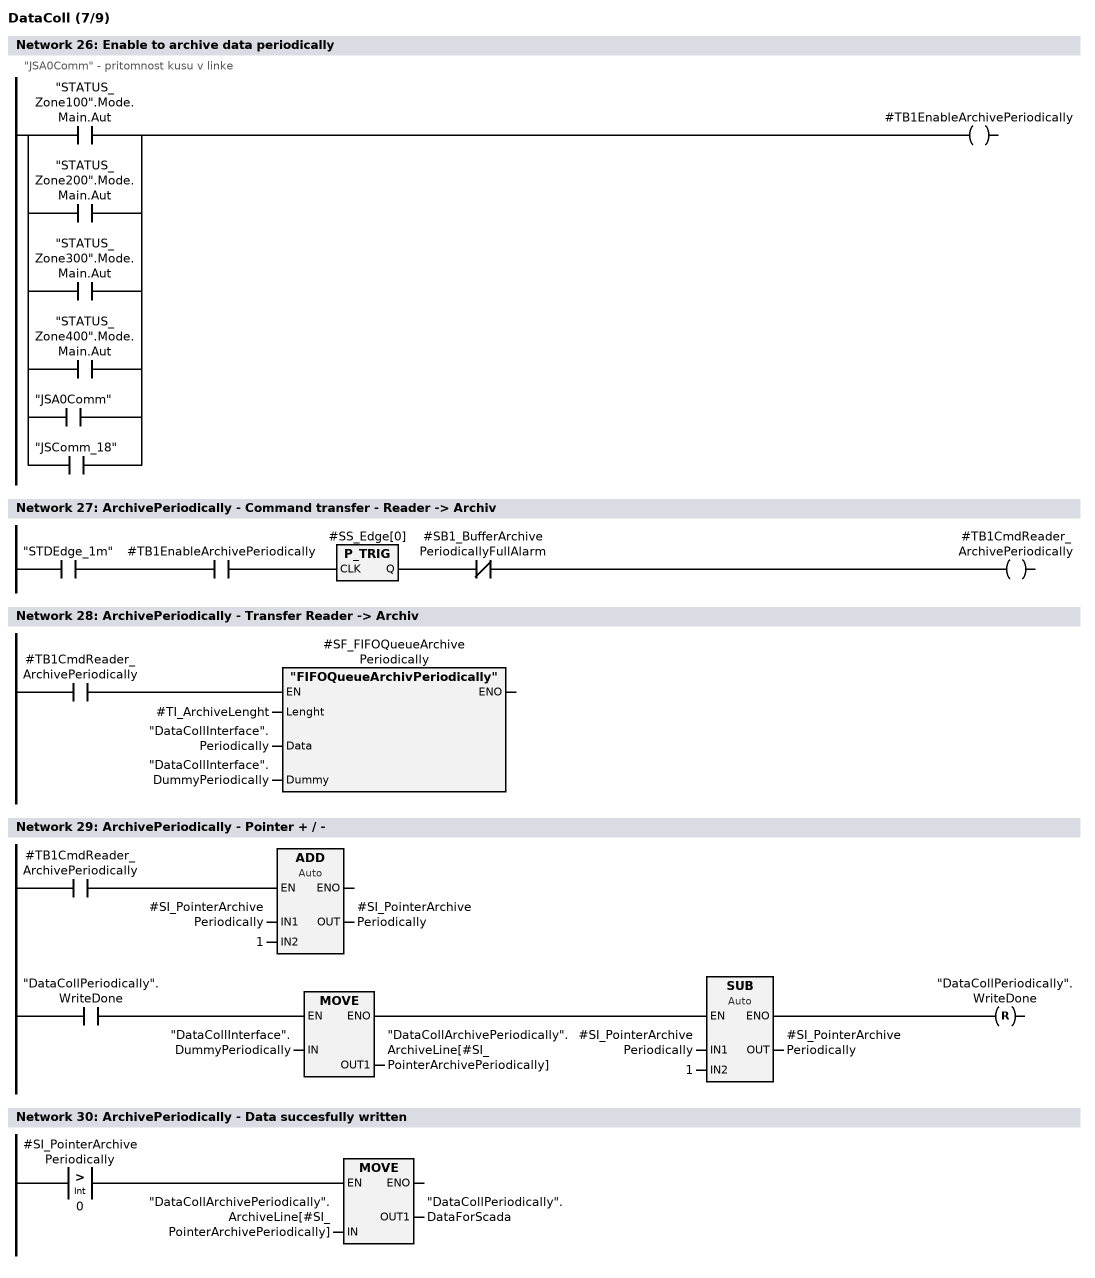
   RUNG wire#powerrail
      Contact( "STATUS_Zone100".Mode.Main.Aut )
      wire#w1
      Coil( #TB1EnableArchivePeriodically )
   END_RUNG
   RUNG wire#powerrail
      Contact( "STATUS_Zone200".Mode.Main.Aut )
   END_RUNG wire#w1
   RUNG wire#powerrail
      Contact( "STATUS_Zone300".Mode.Main.Aut )
   END_RUNG wire#w1
   RUNG wire#powerrail
      Contact( "STATUS_Zone400".Mode.Main.Aut )
   END_RUNG wire#w1
   RUNG wire#powerrail
      Contact( "JSA0Comm" )
   END_RUNG wire#w1
   RUNG wire#powerrail
      Contact( "JSComm_18" )
   END_RUNG wire#w1
   // the same network as SCL:
   #TB1EnableArchivePeriodically := "STATUS_Zone100".Mode.Main.Aut OR "STATUS_Zone200".Mode.Main.Aut OR "STATUS_Zone300".Mode.Main.Aut OR "STATUS_Zone400".Mode.Main.Aut OR "JSA0Comm" OR "JSComm_18";
END_REGION

REGION Network 27: ArchivePeriodically - Command transfer - Reader -> Archiv
   RUNG wire#powerrail
      Contact( "STDEdge_1m" )
      Contact( #TB1EnableArchivePeriodically )
      P_Trig( #SS_Edge[0] )
      I_Contact( #SB1_BufferArchivePeriodicallyFullAlarm )
      Coil( #TB1CmdReader_ArchivePeriodically )
   END_RUNG
   // the same network as SCL:
   #_w1 := "STDEdge_1m" AND #TB1EnableArchivePeriodically;
   #_w2 := #_w1 AND NOT #SS_Edge[0];   // rising edge
   #SS_Edge[0] := #_w1;
   #TB1CmdReader_ArchivePeriodically := #_w2 AND NOT #SB1_BufferArchivePeriodicallyFullAlarm;
END_REGION

REGION Network 28: ArchivePeriodically - Transfer Reader -> Archiv
   RUNG wire#powerrail
      Contact( #TB1CmdReader_ArchivePeriodically )
      #SF_FIFOQueueArchivePeriodically(Lenght := #TI_ArchiveLenght, Data := "DataCollInterface".Periodically, Dummy := "DataCollInterface".DummyPeriodically)
   END_RUNG
   // the same network as SCL:
   IF #TB1CmdReader_ArchivePeriodically THEN
       #SF_FIFOQueueArchivePeriodically(Lenght := #TI_ArchiveLenght,   // "FIFOQueueArchivPeriodically"
                               Data := "DataCollInterface".Periodically,
                               Dummy := "DataCollInterface".DummyPeriodically);
   END_IF;
END_REGION

REGION Network 29: ArchivePeriodically - Pointer + / -
   RUNG wire#powerrail
      Contact( #TB1CmdReader_ArchivePeriodically )
      Add(in1 := #SI_PointerArchivePeriodically, in2 := 1, out => #SI_PointerArchivePeriodically)
   END_RUNG
   RUNG wire#powerrail
      Contact( "DataCollPeriodically".WriteDone )
      Move(in := "DataCollInterface".DummyPeriodically, out1 => "DataCollArchivePeriodically".ArchiveLine[#SI_PointerArchivePeriodically])
      Sub(in1 := #SI_PointerArchivePeriodically, in2 := 1, out => #SI_PointerArchivePeriodically)
      R_Coil( "DataCollPeriodically".WriteDone )
   END_RUNG
   // the same network as SCL:
   IF #TB1CmdReader_ArchivePeriodically THEN
       #SI_PointerArchivePeriodically := #SI_PointerArchivePeriodically + 1;
   END_IF;
   IF "DataCollPeriodically".WriteDone THEN
       "DataCollArchivePeriodically".ArchiveLine[#SI_PointerArchivePeriodically] := "DataCollInterface".DummyPeriodically;
       #SI_PointerArchivePeriodically := #SI_PointerArchivePeriodically - 1;
       "DataCollPeriodically".WriteDone := FALSE;
   END_IF;
END_REGION

REGION Network 30: ArchivePeriodically - Data succesfully written
   RUNG wire#powerrail
      { S7_Templates := "SrcType := Int" } GT_Contact(in1 := #SI_PointerArchivePeriodically, in2 := 0)
      Move(in := "DataCollArchivePeriodically".ArchiveLine[#SI_PointerArchivePeriodically], out1 => "DataCollPeriodically".DataForScada)
   END_RUNG
   // the same network as SCL:
   IF #SI_PointerArchivePeriodically > 0 THEN
       "DataCollPeriodically".DataForScada := "DataCollArchivePeriodically".ArchiveLine[#SI_PointerArchivePeriodically];
   END_IF;
END_REGION

REGION Network 31: ArchivePeriodically - Data ready for SCADA
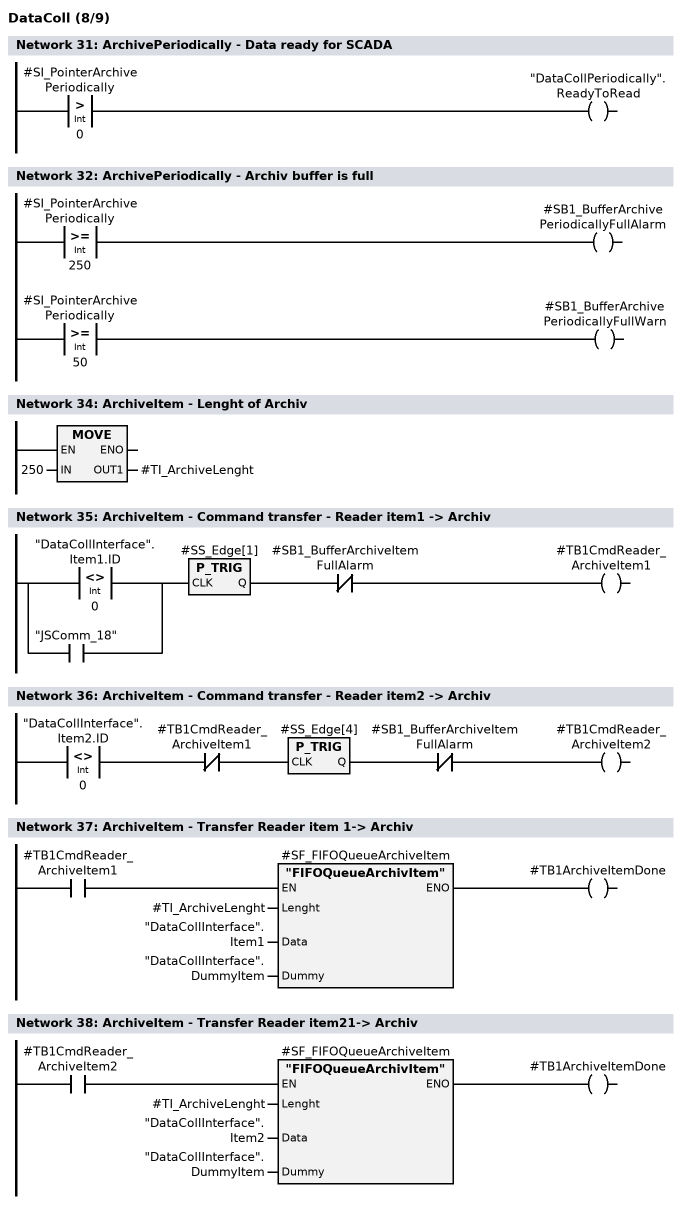
   RUNG wire#powerrail
      { S7_Templates := "SrcType := Int" } GT_Contact(in1 := #SI_PointerArchivePeriodically, in2 := 0)
      Coil( "DataCollPeriodically".ReadyToRead )
   END_RUNG
   // the same network as SCL:
   "DataCollPeriodically".ReadyToRead := #SI_PointerArchivePeriodically > 0;
END_REGION

REGION Network 32: ArchivePeriodically - Archiv buffer is full
   RUNG wire#powerrail
      { S7_Templates := "SrcType := Int" } GE_Contact(in1 := #SI_PointerArchivePeriodically, in2 := 250)
      Coil( #SB1_BufferArchivePeriodicallyFullAlarm )
   END_RUNG
   RUNG wire#powerrail
      { S7_Templates := "SrcType := Int" } GE_Contact(in1 := #SI_PointerArchivePeriodically, in2 := 50)
      Coil( #SB1_BufferArchivePeriodicallyFullWarn )
   END_RUNG
   // the same network as SCL:
   #SB1_BufferArchivePeriodicallyFullAlarm := #SI_PointerArchivePeriodically >= 250;
   #SB1_BufferArchivePeriodicallyFullWarn := #SI_PointerArchivePeriodically >= 50;
END_REGION

REGION Network 33: *************** ArchiveItem ***************
END_REGION

REGION Network 34: ArchiveItem - Lenght of Archiv
   RUNG wire#powerrail
      Move(in := 250, out1 => #TI_ArchiveLenght)
   END_RUNG
   // the same network as SCL:
   #TI_ArchiveLenght := 250;
END_REGION

REGION Network 35: ArchiveItem - Command transfer - Reader item1 -> Archiv
   RUNG wire#powerrail
      { S7_Templates := "SrcType := Int" } NE_Contact(in1 := "DataCollInterface".Item1.ID, in2 := 0)
      wire#w1
      P_Trig( #SS_Edge[1] )
      I_Contact( #SB1_BufferArchiveItemFullAlarm )
      Coil( #TB1CmdReader_ArchiveItem1 )
   END_RUNG
   RUNG wire#powerrail
      Contact( "JSComm_18" )
   END_RUNG wire#w1
   // the same network as SCL:
   #_w1 := ("DataCollInterface".Item1.ID <> 0) OR "JSComm_18";
   #_w2 := #_w1 AND NOT #SS_Edge[1];   // rising edge
   #SS_Edge[1] := #_w1;
   #TB1CmdReader_ArchiveItem1 := #_w2 AND NOT #SB1_BufferArchiveItemFullAlarm;
END_REGION

REGION Network 36: ArchiveItem - Command transfer - Reader item2 -> Archiv
   RUNG wire#powerrail
      { S7_Templates := "SrcType := Int" } NE_Contact(in1 := "DataCollInterface".Item2.ID, in2 := 0)
      I_Contact( #TB1CmdReader_ArchiveItem1 )
      P_Trig( #SS_Edge[4] )
      I_Contact( #SB1_BufferArchiveItemFullAlarm )
      Coil( #TB1CmdReader_ArchiveItem2 )
   END_RUNG
   // the same network as SCL:
   #_w1 := ("DataCollInterface".Item2.ID <> 0) AND NOT #TB1CmdReader_ArchiveItem1;
   #_w2 := #_w1 AND NOT #SS_Edge[4];   // rising edge
   #SS_Edge[4] := #_w1;
   #TB1CmdReader_ArchiveItem2 := #_w2 AND NOT #SB1_BufferArchiveItemFullAlarm;
END_REGION

REGION Network 37: ArchiveItem - Transfer Reader item 1-> Archiv
   RUNG wire#powerrail
      Contact( #TB1CmdReader_ArchiveItem1 )
      #SF_FIFOQueueArchiveItem(Lenght := #TI_ArchiveLenght, Data := "DataCollInterface".Item1, Dummy := "DataCollInterface".DummyItem)
      Coil( #TB1ArchiveItemDone )
   END_RUNG
   // the same network as SCL:
   #SF_FIFOQueueArchiveItem(EN := #TB1CmdReader_ArchiveItem1,   // "FIFOQueueArchivItem"
                           Lenght := #TI_ArchiveLenght,
                           Data := "DataCollInterface".Item1,
                           Dummy := "DataCollInterface".DummyItem,
                           ENO => #_w1);
   #TB1ArchiveItemDone := #_w1;
END_REGION

REGION Network 38: ArchiveItem - Transfer Reader item21-> Archiv
   RUNG wire#powerrail
      Contact( #TB1CmdReader_ArchiveItem2 )
      #SF_FIFOQueueArchiveItem(Lenght := #TI_ArchiveLenght, Data := "DataCollInterface".Item2, Dummy := "DataCollInterface".DummyItem)
      Coil( #TB1ArchiveItemDone )
   END_RUNG
   // the same network as SCL:
   #SF_FIFOQueueArchiveItem(EN := #TB1CmdReader_ArchiveItem2,   // "FIFOQueueArchivItem"
                           Lenght := #TI_ArchiveLenght,
                           Data := "DataCollInterface".Item2,
                           Dummy := "DataCollInterface".DummyItem,
                           ENO => #_w1);
   #TB1ArchiveItemDone := #_w1;
END_REGION

REGION Network 39: ArchiveItem - Position Reader delete data / Position Laser -> Position Reader
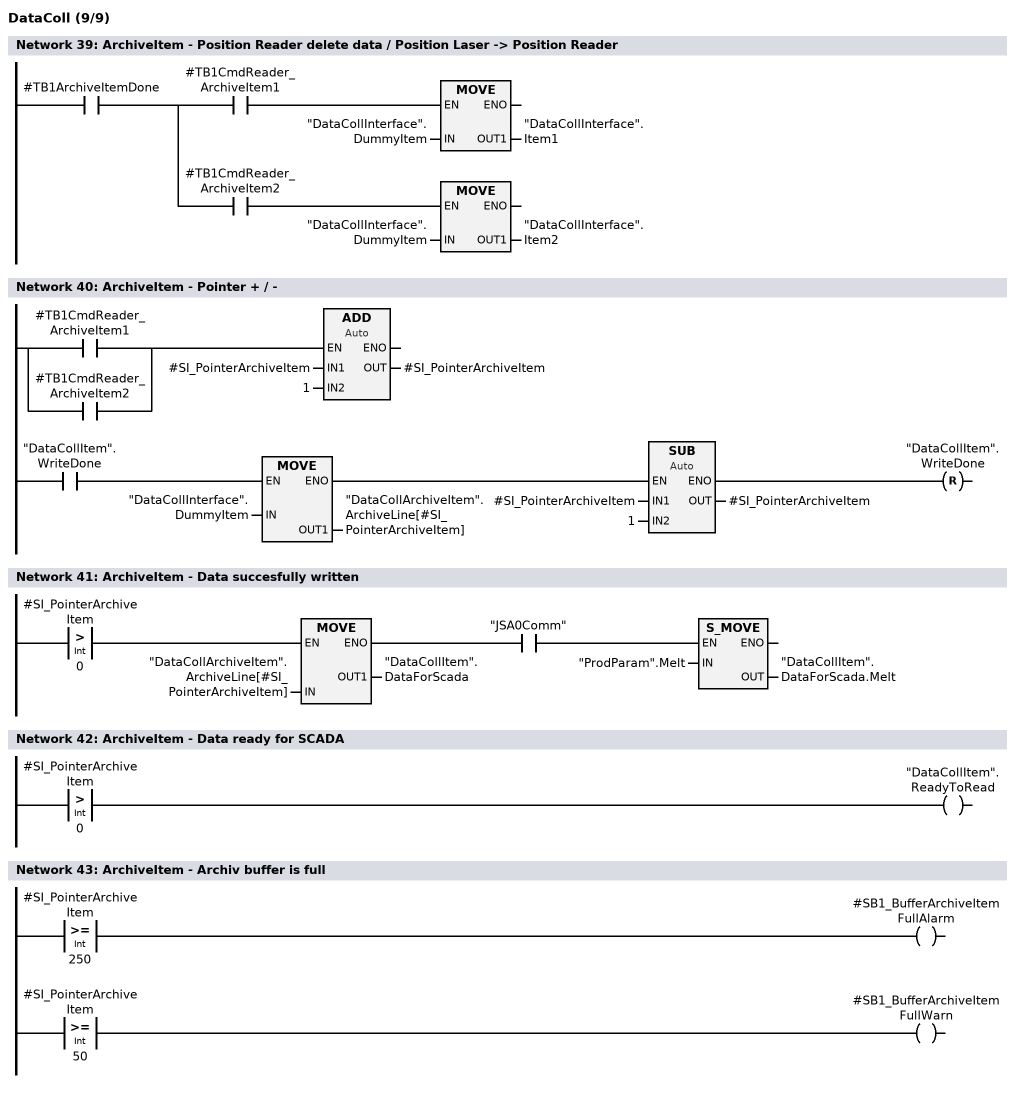
   RUNG wire#powerrail
      Contact( #TB1ArchiveItemDone )
      wire#w1
      Contact( #TB1CmdReader_ArchiveItem1 )
      Move(in := "DataCollInterface".DummyItem, out1 => "DataCollInterface".Item1)
   END_RUNG
   RUNG wire#w1
      Contact( #TB1CmdReader_ArchiveItem2 )
      Move(in := "DataCollInterface".DummyItem, out1 => "DataCollInterface".Item2)
   END_RUNG
   // the same network as SCL:
   IF #TB1ArchiveItemDone AND #TB1CmdReader_ArchiveItem1 THEN
       "DataCollInterface".Item1 := "DataCollInterface".DummyItem;
   END_IF;
   IF #TB1ArchiveItemDone AND #TB1CmdReader_ArchiveItem2 THEN
       "DataCollInterface".Item2 := "DataCollInterface".DummyItem;
   END_IF;
END_REGION

REGION Network 40: ArchiveItem - Pointer + / -
   RUNG wire#powerrail
      Contact( #TB1CmdReader_ArchiveItem1 )
      wire#w1
      Add(in1 := #SI_PointerArchiveItem, in2 := 1, out => #SI_PointerArchiveItem)
   END_RUNG
   RUNG wire#powerrail
      Contact( #TB1CmdReader_ArchiveItem2 )
   END_RUNG wire#w1
   RUNG wire#powerrail
      Contact( "DataCollItem".WriteDone )
      Move(in := "DataCollInterface".DummyItem, out1 => "DataCollArchiveItem".ArchiveLine[#SI_PointerArchiveItem])
      Sub(in1 := #SI_PointerArchiveItem, in2 := 1, out => #SI_PointerArchiveItem)
      R_Coil( "DataCollItem".WriteDone )
   END_RUNG
   // the same network as SCL:
   IF #TB1CmdReader_ArchiveItem1 OR #TB1CmdReader_ArchiveItem2 THEN
       #SI_PointerArchiveItem := #SI_PointerArchiveItem + 1;
   END_IF;
   IF "DataCollItem".WriteDone THEN
       "DataCollArchiveItem".ArchiveLine[#SI_PointerArchiveItem] := "DataCollInterface".DummyItem;
       #SI_PointerArchiveItem := #SI_PointerArchiveItem - 1;
       "DataCollItem".WriteDone := FALSE;
   END_IF;
END_REGION

REGION Network 41: ArchiveItem - Data succesfully written
   RUNG wire#powerrail
      { S7_Templates := "SrcType := Int" } GT_Contact(in1 := #SI_PointerArchiveItem, in2 := 0)
      Move(in := "DataCollArchiveItem".ArchiveLine[#SI_PointerArchiveItem], out1 => "DataCollItem".DataForScada)
      Contact( "JSA0Comm" )
      S_Move(in := "ProdParam".Melt, out => "DataCollItem".DataForScada.Melt)
   END_RUNG
   // the same network as SCL:
   #_w1 := #SI_PointerArchiveItem > 0;
   IF #_w1 THEN
       "DataCollItem".DataForScada := "DataCollArchiveItem".ArchiveLine[#SI_PointerArchiveItem];
   END_IF;
   IF #_w1 AND "JSA0Comm" THEN "DataCollItem".DataForScada.Melt := "ProdParam".Melt; END_IF;
END_REGION

REGION Network 42: ArchiveItem - Data ready for SCADA
   RUNG wire#powerrail
      { S7_Templates := "SrcType := Int" } GT_Contact(in1 := #SI_PointerArchiveItem, in2 := 0)
      Coil( "DataCollItem".ReadyToRead )
   END_RUNG
   // the same network as SCL:
   "DataCollItem".ReadyToRead := #SI_PointerArchiveItem > 0;
END_REGION

REGION Network 43: ArchiveItem - Archiv buffer is full
   RUNG wire#powerrail
      { S7_Templates := "SrcType := Int" } GE_Contact(in1 := #SI_PointerArchiveItem, in2 := 250)
      Coil( #SB1_BufferArchiveItemFullAlarm )
   END_RUNG
   RUNG wire#powerrail
      { S7_Templates := "SrcType := Int" } GE_Contact(in1 := #SI_PointerArchiveItem, in2 := 50)
      Coil( #SB1_BufferArchiveItemFullWarn )
   END_RUNG
   // the same network as SCL:
   #SB1_BufferArchiveItemFullAlarm := #SI_PointerArchiveItem >= 250;
   #SB1_BufferArchiveItemFullWarn := #SI_PointerArchiveItem >= 50;
END_REGION
END_FUNCTION_BLOCK
